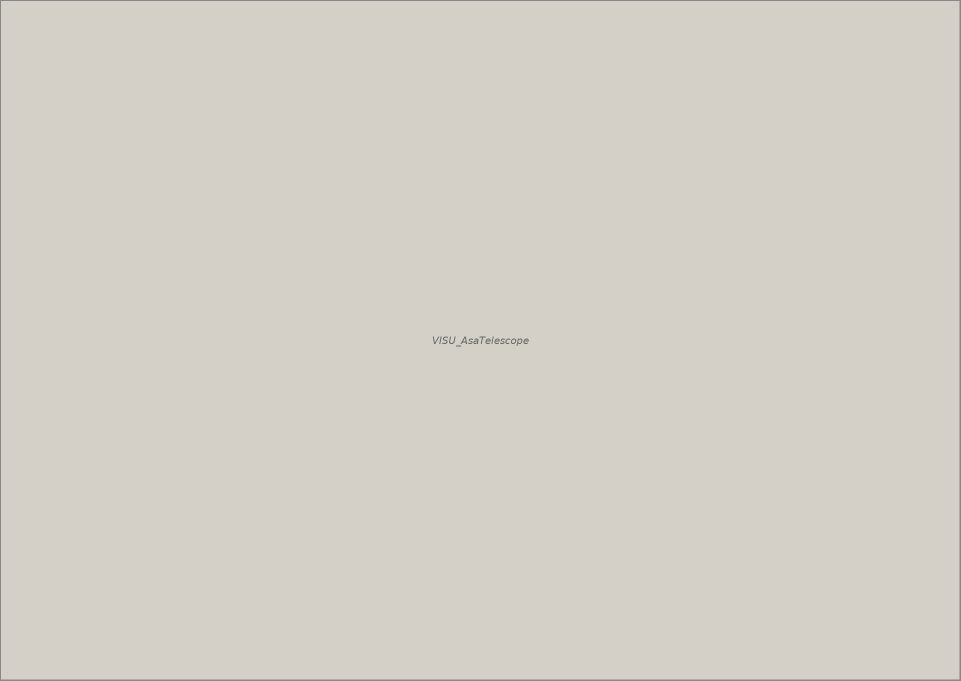
VISUALIZATION VISU_MAIN  // 961x681
    Frame (0,0 961x681)
        shows VISU_AsaTelescope(fbInstance := MAIN.fbTelescope)
END_VISUALIZATION

(* stored: Version 1.1.0.1, ProductVersion 3.1.4024.12
   Visu VISU_MAIN: Id {6a0ea8df-ebb3-410b-b05e-aa4b69f614d6} *)
